(* Schneider Machine Expert - Basic project grafcet, file version 3.0.0.0 *)
(* ProjectInformations: Name=Nuovo progetto *)

HARDWARE
  Cpu 0: TM221M16R/G
  EthernetConfiguration: NetworkName=M221, IpAllocationMode=FixedAddress, IpAddress=0.0.0.0, SubnetMask=0.0.0.0
  SerialLineConfiguration: Baud=Baud19200, Parity=ParityEven, DataBits=DataBits8, StopBits=StopBits1, PhysicalMedium=PhysicalMediumRs485, TransmissionMode=TransmissionModeModbusRtu, SlaveId=1, Addressing=SlaveAddressing
  MastTask: UsePeriodScanMode=false, PeriodScan=100
  FastTask: Period=255
  CpuBehavior: StartingMode=StartAsPreviousState, AutoSaveRamOnEeprom=true, WatchdogPeriod=250

SYMBOLS  (address, symbol, comment, settings)
  %I0.0     BTN_START

GRAFCET Grafcet POU
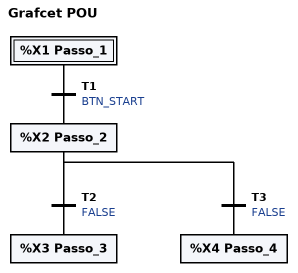
  INITIAL_STEP %X1  (* Passo_1 *)
  STEP %X2  (* Passo_2 *)
  STEP %X3  (* Passo_3 *)
  STEP %X4  (* Passo_4 *)
  TRANSITION T1 FROM %X1 TO %X2 := BTN_START;
  TRANSITION T2 FROM %X2 TO %X3 := FALSE;
  TRANSITION T3 FROM %X2 TO %X4 := FALSE;

STEP %X2 Passo_2
  (* SectionNumber=0, StepNumber=2 *)

// Rung 0
  LD

TRANSITION T1 (%X1 -> %X2) 
  (* SectionNumber=0 *)

// Rung 1: Tr1
  LD %I0.0                (* BTN_START *)
  ENDT
  // as ST:
  //   TRANSITION := BTN_START;

TRANSITION T2 (%X2 -> %X3) 
  (* SectionNumber=0 *)

// Rung 2: Tr2
  LD 0
  ENDT
  // as ST:
  //   TRANSITION := FALSE;

TRANSITION T3 (%X2 -> %X4) 
  (* SectionNumber=0 *)

// Rung 3: Tr3
  LD 0
  ENDT
  // as ST:
  //   TRANSITION := FALSE;
